# EPICS autosave request: iocBoot/iocTomoScan_32ID_STEP/auto_settings.req
file "tomoScan_settings.req", P=$(P), R=$(R)
file "tomoScan_PSO_settings.req", P=$(P), R=$(R)
file "tomoScan_32ID_settings.req", P=$(P), R=$(R)
